// TIA Portal V19 export
DATA_BLOCK "JB_PERS"   // DB64
// stored: MemoryReserve 100
   VAR RETAIN
      PersistentValues : Struct
         Data : Struct
            WeldingSetUp : "JB_WeldingSetUp";
            ClampEntryClosed : Bool := FALSE;
            ClampExitClosed : Bool := FALSE;
         END_STRUCT;
         Torch : Struct
            MeasureTorchHolder : LReal := 70.0;   // Distance from sliding block & torch holder
            InhibitWeld_Pos : LReal := 0.0;
            InhibitWeld_Window : LReal := 0.0;   // if > 0 the ihhibit is enabled
            Parking_Pos : LReal := -310.0;
            WeldingUseLocalData : Bool := FALSE;   // TRUE = USE LOCAL DATA / FALSE = USE PROFILE DATA
            Cycle_HighSpeed : LReal := 100.0;   // 0..100%
            Cycle_LowSpeed : LReal := 50.0;   // 0..100%
         END_STRUCT;
         TorchAx : "Positioning_DOL_Machine_Par";
         TorchAx_Pers { ExternalAccessible := 'False'; ExternalVisible := 'False'; ExternalWritable := 'False'} : "Positioning_DOL_Machine_Pers_Data";
         TorchEnc : "PosFbk_RTN";
         PinchRoll_Feed : "SpeedMachine_Par";
         Aspiratore_TimeOff { S7_SetPoint := 'True'} : Time;
      END_STRUCT;
   END_VAR
BEGIN
   PersistentValues.Data.WeldingSetUp.MaterialWidth := 220.0;
   PersistentValues.Data.WeldingSetUp.MeasureSheetEdgeReference := 0.0;
   PersistentValues.Data.WeldingSetUp.WeldingDirection := TRUE;
   PersistentValues.Data.WeldingSetUp.CorrStartWelding := 5.0;
   PersistentValues.Data.WeldingSetUp.CorrStopWelding := 5.0;
   PersistentValues.TorchAx.PosTolerance := 0.3;
   PersistentValues.TorchAx.Minus_Limit := -320.0;
   PersistentValues.TorchAx.Plus_Limit := 310.0;
   PersistentValues.TorchAx.PreCutOff := 0.2;
   PersistentValues.TorchAx.PreEndLowSpeed := 2.0;
   PersistentValues.TorchAx.PreEndMedSpeed := 5.0;
   PersistentValues.TorchAx.LowSpeed := 15.0;
   PersistentValues.TorchAx.MedSpeed := 70.0;
   PersistentValues.TorchAx.HighSpeed := 70.0;
   PersistentValues.TorchAx.Man_Speed := 100.0;
   PersistentValues.TorchAx_Pers.AxisHomed := TRUE;
   PersistentValues.TorchEnc.Preset.Pulses := 0;
   PersistentValues.TorchEnc.Preset.Units := -309.48;
   PersistentValues.TorchEnc.Config.Resolution := 5.0;
   PersistentValues.PinchRoll_Feed.Man.VelBwd := 5000.0;
   PersistentValues.PinchRoll_Feed.Man.VelFwdHigh := 5000.0;
   PersistentValues.PinchRoll_Feed.Man.VelFwdLow := 2000.0;
   PersistentValues.PinchRoll_Feed.Man.Acc := 1000.0;
   PersistentValues.PinchRoll_Feed.Man.Dec := 1000.0;
   PersistentValues.PinchRoll_Feed.Man.DelayChangeVel := T#5S;
END_DATA_BLOCK
